TYPE ST_SubProgramTable :
STRUCT
	AxisTable						: ARRAY [1..No, 0..59999] OF LREAL;
	AirTable							: ARRAY [1..AirNo, 0..59999] OF BOOL;
	ExFSpdUpTable					: ARRAY [0..59999] OF BOOL;
END_STRUCT
END_TYPE

(* stored: Version 1.1.0.1, ProductVersion 3.1.4024.9
   DUT ST_SubProgramTable: Id {e3d9b176-2892-42a3-881c-fa651d5f1be7} *)
